// This function has been automatically generated from the project information.
{attribute 'signature_flag' := '1073741824'}
{attribute 'TcGenerated'}
{attribute 'no-analysis'}
FUNCTION F_GetTitle : WSTRING
VAR_INPUT
	
END_VAR

F_GetTitle := "FsCommon";

END_FUNCTION

(* stored: Version 1.1.0.1
   POU F_GetTitle: Id {00d38eff-2f4b-07d9-3abb-6c10748da9b8}, SpecialFunc None *)
